(* CoDeSys 2.3 export: FB_EMPTYBLOCK.EXP *)

(* POU FB_EmptyBlock, ST *)
FUNCTION_BLOCK FB_EmptyBlock
VAR_INPUT
END_VAR
VAR_OUTPUT
END_VAR
VAR
END_VAR
;
END_FUNCTION_BLOCK
